{attribute 'Tc2GvlVarNames'}
VAR_GLOBAL
END_VAR

(* stored: Version 1.1.0.1, ProductVersion 3.1.4018.9
   GVL Global_Variables: Id {918b328c-1402-466d-aff2-e349ff1e6cb1} *)
